PROGRAM MAIN
VAR
	inputDigSens1 AT %I*: BOOL;
	inputDigSens2 AT %I*: BOOL;
	nichtGutBit:BOOL:=FALSE;
	allesGutBit:BOOL;
	
END_VAR

// the two optical sensors can never be zero at the same time because Pilz overspeed will trip
IF NOT inputDigSens1 AND NOT inputDigSens2 THEN
	nichtGutBit:=TRUE;
END_IF
allesGutBit:=NOT nichtGutBit;

END_PROGRAM

(* stored: Version 1.1.0.1, ProductVersion 3.1.4022.6
   POU MAIN: Id {e3706b08-6154-42eb-8c8a-7893886a10c9}, SpecialFunc None *)
